// Mitsubishi GX Works2 project: yudomotor   PLC: Q03UDV

PROGRAM MAIN
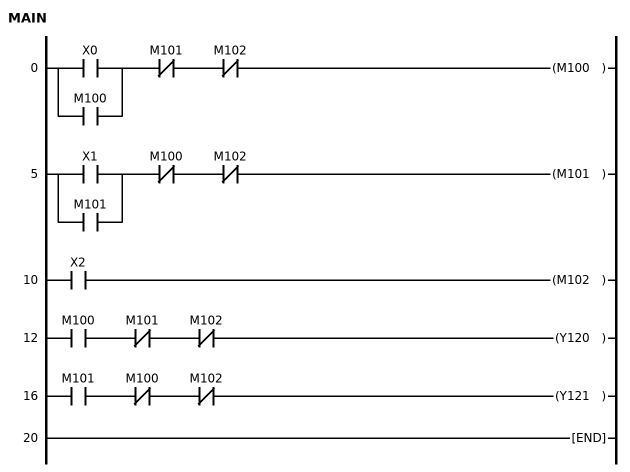
0     LD      X0
      OR      M100
      ANI     M101
      ANI     M102
      OUT     M100
5     LD      X1
      OR      M101
      ANI     M100
      ANI     M102
      OUT     M101
10    LD      X2
      OUT     M102
12    LD      M100
      ANI     M101
      ANI     M102
      OUT     Y120
16    LD      M101
      ANI     M100
      ANI     M102
      OUT     Y121
20    END
END_PROGRAM
